% RSLogix 500 project heater_pid.RSS, saved by version 8.30.00.16 %
PROJECT "UNTITLED"    % processor: Bul.1763 MicroLogix 1100 Series B %

PROGRAM FILES
  LAD 2 "MAIN"  5 rungs

DATA FILES
  O0 OUTPUT  5 elements
  I1 INPUT  7 elements
  S2 STATUS  66 elements
  B3 BINARY  1 elements
  T4 TIMER  1 elements
  C5 COUNTER  1 elements
  R6 CONTROL  1 elements
  N7 INTEGER  1 elements
  F8 FLOAT  1 elements

LADDER 2 "MAIN"
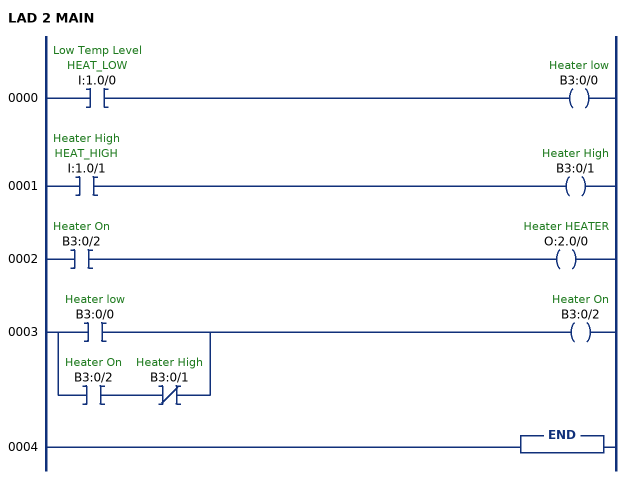
% Rung: 0 %
SOR XIC I:1.0/0 OTE B3:0/0 EOR
%   I:1.0/0  HEAT_LOW  "Low Temp Level" %
%   B3:0/0  "Heater low" %
% Rung: 1 %
SOR XIC I:1.0/1 OTE B3:0/1 EOR
%   I:1.0/1  HEAT_HIGH  "Heater High" %
%   B3:0/1  "Heater High" %
% Rung: 2 %
SOR XIC B3:0/2 OTE O:2.0/0 EOR
%   B3:0/2  "Heater On" %
%   O:2.0/0  HEATER  "Heater" %
% Rung: 3 %
SOR BST XIC B3:0/0 NXB XIC B3:0/2 XIO B3:0/1 BND OTE B3:0/2 EOR
%   B3:0/0  "Heater low" %
%   B3:0/2  "Heater On" %
%   B3:0/1  "Heater High" %
% Rung: 4 %
SOR END EOR

OTHER DOCUMENTED ADDRESSES
  I:2.0/0  L_HEAT  "Heater Low"
  I:3.0/0  "Heater Low Limit"
  I:3.0/1  "Heater High Limit"
  O:3.0  "Heater On"
  O:3.0/0  HEATER_ON  "Heater On"
  T4:0  "Heat Low Timer"
  T4:0/DN  "Timer for Heater DN"
  T4:1  "Heat High"
  T4:1/DN  "Heater Off"
  U:3  "IO"
  U:4  "CONTROLS"
